FUNCTION_BLOCK CHECKPOINT_DISCOVERY_CAT_HMI (* Service Interface Function Block Type *)
  (* Standard: 61499-2 *)
  (* Version 0.0, 1/24/2023, Dmitrii, Flexbridge AB, template *)
  PACKAGE UAO.Hackathon;
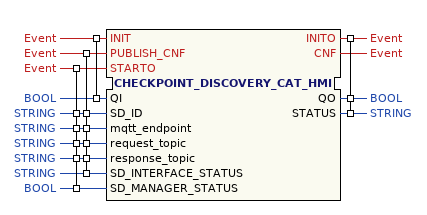
  EVENT_INPUT
    INIT WITH QI;
    PUBLISH_CNF WITH SD_ID, mqtt_endpoint, request_topic, response_topic, SD_INTERFACE_STATUS;
    STARTO WITH SD_ID, mqtt_endpoint, request_topic, response_topic, SD_MANAGER_STATUS;
  END_EVENT
  EVENT_OUTPUT
    INITO WITH QO, STATUS;
    CNF;
  END_EVENT
  VAR_INPUT
    QI : BOOL;
    SD_ID : STRING;
    mqtt_endpoint : STRING;
    request_topic : STRING;
    response_topic : STRING;
    SD_INTERFACE_STATUS : STRING;
    SD_MANAGER_STATUS : BOOL;
  END_VAR
  VAR_OUTPUT
    QO : BOOL; (* Event Output Qualifier *)
    STATUS : STRING; (* Service Status *)
  END_VAR
  SERVICE /
    SEQUENCE 
    END_SEQUENCE
  END_SERVICE
END_FUNCTION_BLOCK
